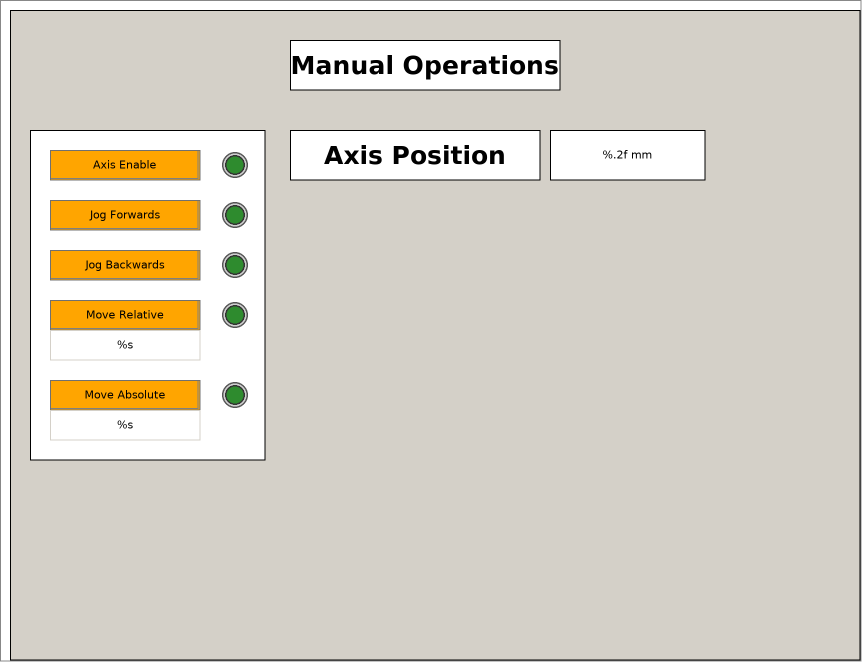
VISUALIZATION Manual_Operations  // 862x662
    RoundedRectangle (10,10 850x650)
    Rectangle (30,130 235x330)
    RoundedRectangle (290,40 270x50), "Manual Operations"
    Button (50,200 150x30), "Jog Forwards"
        OnMouseDown: toggle MAIN.bJogForwards
        OnMouseUp: toggle MAIN.bJogForwards
        OnMouseUp: execute { MAIN.bEnableAxis_1 := TRUE }
    Lamp1 (220,200 30x30), variable: MAIN.bJogForwards, style: Lamp-Lamp1-Green
    Button (50,150 150x30), "Axis Enable"
        toggle MAIN.bEnableAxis_1
    Lamp1 (220,150 30x30), variable: MAIN.mcPower_1.Enable, style: Lamp-Lamp1-Green
    Button (50,250 150x30), "Jog Backwards"
        OnMouseDown: toggle MAIN.bJogBackwards
        OnMouseUp: toggle MAIN.bJogBackwards
        OnMouseUp: execute { MAIN.bEnableAxis_1 := TRUE }
    Lamp1 (220,250 30x30), variable: MAIN.bJogBackwards, style: Lamp-Lamp1-Green
    Button (50,300 150x30), "Move Relative"
        toggle MAIN.bRelMove p2164770859=TRUE
    Lamp1 (220,300 30x30), variable: MAIN.mcMoveRel_1.Active, style: Lamp-Lamp1-Green
    Textfield (50,330 150x30), "%s", text variable: MAIN.fRelDistance
        OnMouseClick: write the text variable via VisuDialogs.Numpad, min -100, max 100, format Relative Move Distance
    Button (50,380 150x30), "Move Absolute"
        toggle MAIN.bAbsMove p2164770859=TRUE
    Lamp1 (220,380 30x30), variable: MAIN.mcMoveAbs_1.Active, style: Lamp-Lamp1-Green
    Textfield (50,410 150x30), "%s", text variable: MAIN.fAbsPos_1
        OnMouseClick: write the text variable via VisuDialogs.Numpad, min -100, max 100, format Relative Move Distance
    RoundedRectangle (290,130 250x50), "Axis Position"
    RoundedRectangle (550,130 155x50), "%.2f mm", text variable: GVL.stAxis_1.NcToPlc.SetPos
END_VISUALIZATION

(* stored: Version 1.1.0.1, ProductVersion 3.1.4024.0
   Visu Manual_Operations: Id {42bf85bb-a55c-43f2-b75e-c1688e11f525} *)
